Staubli VAL3: OnStartup.pgx

public program OnStartup()
begin
  //
  // use to create custom tasks
  // taskCreate...
  //
end
